// Mitsubishi GX Developer project: Conter_Up   PLC: FX3U

PROGRAM MAIN
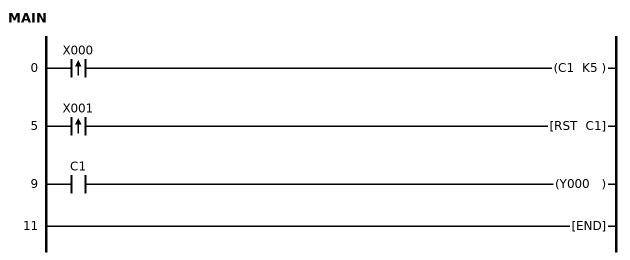
0     LDP     X000
      OUT     C1 K5
5     LDP     X001
      RST     C1
9     LD      C1
      OUT     Y000
11    END
END_PROGRAM
